// TIA Portal V16 export
// export: Created 2021-11-12T13:32:58.1508779Z, ExportSetting WithDefaults, DisplayName Totally Integrated Automation Portal, DisplayVersion V16 Update 3, DisplayName TIA Portal Version Control Interface, DisplayVersion V16 Update 2, DisplayName TIA Portal Openness, DisplayVersion V16 Update 3, DisplayName SINAMICS Startdrive Advanced, DisplayVersion V16 Update 5, DisplayName SINAMICS Startdrive G130, G150, S120, S150, SINAMICS MV, S210, DisplayVersion V16 Update 5, DisplayName SINAMICS Startdrive G110M, G120, G120C, G120D, G120P, G115D, DisplayVersion V16 Update 5, DisplayName STEP 7 Professional, DisplayVersion V16 Update 3, DisplayName STEP 7 Safety, DisplayVersion V16, DisplayName WinCC UA Professional, DisplayVersion V16 Update 3
DATA_BLOCK "IDB_Zone300"   // DB193
{ DB_Accessible_From_OPC_UA := 'FALSE' }
VERSION : 0.1
// stored: AutoNumber true, DBAccessibleFromOPCUA false, InstanceOfName Zone300, InstanceOfType FB
"Zone300"
   // VAR
   //    SF_ZoneMode { S7_SetPoint := 'True'} : "STD_Zone";
   //    SF_Station320Mode { S7_SetPoint := 'True'} : "STD_Station";
   //    SF_Station310Mode { S7_SetPoint := 'True'} : "STD_Station";
   //    SF_Station330Mode { S7_SetPoint := 'True'} : "STD_Station";
   //    SF_StationBSN4Mode { S7_SetPoint := 'True'} : "STD_Station";
   //    SF_StationBSN5Mode { S7_SetPoint := 'True'} : "STD_Station";
   //    SF_CameraLights { S7_SetPoint := 'True'} : "STD_OnOff";
   //    SF_CameraLights_1 { S7_SetPoint := 'True'} : "STD_OnOff";
   //    SS_Edge { S7_SetPoint := 'True'} : Array[0..100] of Bool;
   // END_VAR
BEGIN
END_DATA_BLOCK
